// TIA Portal V17 program export: 0 tag tables, 0 data types, 1 data blocks, 3 code blocks (in call order from the OBs), 0 instance data blocks

DATA_BLOCK "DB_GlobalData"   // DB1
{ S7_Optimized_Access := 'TRUE' }
VERSION : 0.1
// stored: AutoNumber true, DBAccessibleFromOPCUA true, DataBlockType GlobalDB, IsIECCheckEnabled false, IsRetainMemResEnabled false, MemoryReserve 100
   VAR
      Start_Button { ExternalWritable := 'False'} : Bool;   // Start button input
      Stop_Button : Bool;   // Stop button input
      Emergency_Stop : Bool;   // Emergency stop input
      Motor_Running : Bool;   // Motor running status
      Motor_Speed : Real := 0.0;   // Current motor speed RPM
      Speed_Setpoint : Real := 1500.0;   // Desired motor speed RPM
      Temperature : Real := 25.0;   // Motor temperature in Celsius
      RunTime_Hours : DInt := 0;   // Total runtime hours
      Alarm_Active : Bool;   // Alarm status flag
      Alarm_Code : Word := 16#0000;   // Alarm code identifier
   END_VAR
BEGIN
END_DATA_BLOCK

ORGANIZATION_BLOCK "Main"   // OB1, LAD, ProgramCycle
{ S7_Optimized_Access := 'TRUE' }
VERSION : 0.1
// stored: AutoNumber true, IsIECCheckEnabled false
   VAR_INPUT
      Initial_Call : Bool;
      Remanence : Bool;
   END_VAR
BEGIN

REGION Network 1: Motor Control Logic
   // Start motor when button pressed
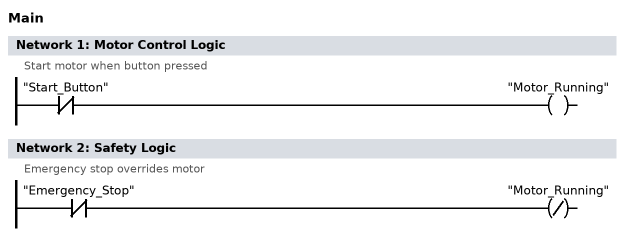
   RUNG wire#powerrail
      I_Contact( "Start_Button" )
      Coil( "Motor_Running" )
   END_RUNG
   // the same network as SCL:
   "Motor_Running" := NOT "Start_Button";
END_REGION

REGION Network 2: Safety Logic
   // Emergency stop overrides motor
   RUNG wire#powerrail
      I_Contact( "Emergency_Stop" )
      I_Coil( "Motor_Running" )
   END_RUNG
   // the same network as SCL:
   "Motor_Running" := NOT (NOT "Emergency_Stop");
END_REGION
END_ORGANIZATION_BLOCK

FUNCTION_BLOCK "FB_PID_Controller"   // FB20, SCL
{ S7_Optimized_Access := 'TRUE' }
AUTHOR : Control Systems
FAMILY : Controllers
NAME : PID Controller
VERSION : 2.1
// stored: AutoNumber true, IsIECCheckEnabled true
   VAR_INPUT
      Setpoint : Real;
      ProcessValue : Real;
      Kp : Real;
      Ki : Real;
      Kd : Real;
      Enable : Bool;
   END_VAR
   VAR_OUTPUT
      ControlOutput : Real;
      Error : Real;
   END_VAR
   VAR
      IntegralSum : Real;
      LastError : Real;
      Initialized : Bool;
   END_VAR
   VAR_TEMP
      PropTerm : Real;
      IntTerm : Real;
      DiffTerm : Real;
   END_VAR
BEGIN
// PID Control Algorithm
// PID controller with anti-windup protection
   // PID Controller Implementation
   IF #Enable THEN
       // Calculate error
       #Error := #Setpoint - #ProcessValue;

       // Proportional term
       #PropTerm := #Kp * #Error;

       // Integral term
       #IntegralSum := #IntegralSum + #Error;
       #IntTerm := #Ki * #IntegralSum;

       // Derivative term
       IF #Initialized THEN
           #DiffTerm := #Kd * (#Error - #LastError);
       ELSE
           #DiffTerm := 0.0;
           #Initialized := TRUE;
       END_IF;

       // Calculate control output
       #ControlOutput := #PropTerm + #IntTerm + #DiffTerm;

       // Anti-windup
       IF #ControlOutput > 100.0 THEN
           #ControlOutput := 100.0;
           #IntegralSum := #IntegralSum - #Error;
       ELSIF #ControlOutput < 0.0 THEN
           #ControlOutput := 0.0;
           #IntegralSum := #IntegralSum - #Error;
       END_IF;

       // Save error for next cycle
       #LastError := #Error;
   ELSE
       // Reset controller
       #ControlOutput := 0.0;
       #IntegralSum := 0.0;
       #LastError := 0.0;
       #Initialized := FALSE;
   END_IF;
END_FUNCTION_BLOCK

FUNCTION "FC_MotorControl" : Void   // FC10, SCL
{ S7_Optimized_Access := 'TRUE' }
AUTHOR : Engineering Team
FAMILY : Motors
NAME : Motor Control Function
VERSION : 1.0
// stored: AutoNumber true, IsIECCheckEnabled true
   VAR_INPUT
      Start : Bool;
      Stop : Bool;
      Speed_Setpoint : Real;
   END_VAR
   VAR_OUTPUT
      Motor_On : Bool;
      Current_Speed : Real;
   END_VAR
   VAR_TEMP
      temp_speed : Real;
   END_VAR
BEGIN
// Motor Control
// Main motor control with speed ramping
   // Motor Control Logic
   IF #Start AND NOT #Stop THEN
       #Motor_On := TRUE;
       #temp_speed := #Speed_Setpoint;

       // Ramp up speed
       IF #Current_Speed < #temp_speed THEN
           #Current_Speed := #Current_Speed + 10.0;
           IF #Current_Speed > #temp_speed THEN
               #Current_Speed := #temp_speed;
           END_IF;
       END_IF;
   ELSE
       #Motor_On := FALSE;
       // Ramp down speed
       IF #Current_Speed > 0.0 THEN
           #Current_Speed := #Current_Speed - 10.0;
           IF #Current_Speed < 0.0 THEN
               #Current_Speed := 0.0;
           END_IF;
       END_IF;
   END_IF;
END_FUNCTION
